(* IEC 61131-3 sources: iolink/src/types/serialization/Simatic.Ax.IOLink/BigEndian, 4 files *)

(* ---- BlockDefinition.st ---- *)
// This is generated code. *** DO NOT MODIFY ***

NAMESPACE Simatic.Ax.iolink
FUNCTION SerializeBig : UDINT
    VAR_INPUT
        offset : UDINT;
    END_VAR
    VAR_IN_OUT
        value : BlockDefinition;
        buffer : ARRAY[*] OF BYTE;
    END_VAR
    SerializeBig := offset;
    SerializeBig := System.Serialization.SerializeBig(offset := SerializeBig, value := value.BlockNoDefinition, buffer := buffer);
    SerializeBig := System.Serialization.SerializeBig(offset := SerializeBig, value := value.Channel, buffer := buffer);
    SerializeBig := System.Serialization.SerializeBig(offset := SerializeBig, value := value.BlockType, buffer := buffer);
    SerializeBig := System.Serialization.SerializeBig(offset := SerializeBig, value := value.Version, buffer := buffer);
    SerializeBig := System.Serialization.SerializeBig(offset := SerializeBig, value := value.ByteLength, buffer := buffer);
END_FUNCTION

FUNCTION DeserializeBig : UDINT
    VAR_INPUT
        offset : UDINT;
        buffer : ARRAY[*] OF BYTE;
    END_VAR
    VAR_IN_OUT
        value : BlockDefinition;
    END_VAR
    DeserializeBig := offset;
    DeserializeBig := System.Serialization.DeserializeBig(offset := DeserializeBig, value := value.BlockNoDefinition, buffer := buffer);
    DeserializeBig := System.Serialization.DeserializeBig(offset := DeserializeBig, value := value.Channel, buffer := buffer);
    DeserializeBig := System.Serialization.DeserializeBig(offset := DeserializeBig, value := value.BlockType, buffer := buffer);
    DeserializeBig := System.Serialization.DeserializeBig(offset := DeserializeBig, value := value.Version, buffer := buffer);
    DeserializeBig := System.Serialization.DeserializeBig(offset := DeserializeBig, value := value.ByteLength, buffer := buffer);
END_FUNCTION
END_NAMESPACE

(* ---- DeviceHeader.st ---- *)
// This is generated code. *** DO NOT MODIFY ***

NAMESPACE Simatic.Ax.iolink
FUNCTION SerializeBig : UDINT
    VAR_INPUT
        offset : UDINT;
    END_VAR
    VAR_IN_OUT
        value : DeviceHeader;
        buffer : ARRAY[*] OF BYTE;
    END_VAR
    SerializeBig := offset;
    SerializeBig := System.Serialization.SerializeBig(offset := SerializeBig, value := value.crc32, buffer := buffer);
    SerializeBig := System.Serialization.SerializeBig(offset := SerializeBig, value := value.SourceDestAddress, buffer := buffer);
    SerializeBig := System.Serialization.SerializeBig(offset := SerializeBig, value := value.TypeIdent, buffer := buffer);
    SerializeBig := System.Serialization.SerializeBig(offset := SerializeBig, value := value.ByteLength, buffer := buffer);
    SerializeBig := System.Serialization.SerializeBig(offset := SerializeBig, value := value.NoOfBlocks, buffer := buffer);
END_FUNCTION

FUNCTION DeserializeBig : UDINT
    VAR_INPUT
        offset : UDINT;
        buffer : ARRAY[*] OF BYTE;
    END_VAR
    VAR_IN_OUT
        value : DeviceHeader;
    END_VAR
    DeserializeBig := offset;
    DeserializeBig := System.Serialization.DeserializeBig(offset := DeserializeBig, value := value.crc32, buffer := buffer);
    DeserializeBig := System.Serialization.DeserializeBig(offset := DeserializeBig, value := value.SourceDestAddress, buffer := buffer);
    DeserializeBig := System.Serialization.DeserializeBig(offset := DeserializeBig, value := value.TypeIdent, buffer := buffer);
    DeserializeBig := System.Serialization.DeserializeBig(offset := DeserializeBig, value := value.ByteLength, buffer := buffer);
    DeserializeBig := System.Serialization.DeserializeBig(offset := DeserializeBig, value := value.NoOfBlocks, buffer := buffer);
END_FUNCTION
END_NAMESPACE

(* ---- LIOLink_typeJob.st ---- *)
// This is generated code. *** DO NOT MODIFY ***

NAMESPACE Simatic.Ax.IOLink
FUNCTION SerializeBig : UDINT
    VAR_INPUT
        offset : UDINT;
    END_VAR
    VAR_IN_OUT
        value : LIOLink_typeJob;
        buffer : ARRAY[*] OF BYTE;
    END_VAR
    VAR_TEMP
        i : DINT;
    END_VAR
    SerializeBig := offset;
    SerializeBig := System.Serialization.SerializeBig(offset := SerializeBig, value := value.ExtendedFunctionNum, buffer := buffer);
    SerializeBig := System.Serialization.SerializeBig(offset := SerializeBig, value := value.Options, buffer := buffer);
    SerializeBig := System.Serialization.SerializeBig(offset := SerializeBig, value := value.SequenceNo, buffer := buffer);
    FOR i := DINT#0 TO DINT#233 DO
        SerializeBig := System.Serialization.SerializeBig(offset := SerializeBig, value := value.payload[i], buffer := buffer);
    END_FOR;
END_FUNCTION

FUNCTION DeserializeBig : UDINT
    VAR_INPUT
        offset : UDINT;
        buffer : ARRAY[*] OF BYTE;
    END_VAR
    VAR_IN_OUT
        value : LIOLink_typeJob;
    END_VAR
    VAR_TEMP
        i : DINT;
    END_VAR
    DeserializeBig := offset;
    DeserializeBig := System.Serialization.DeserializeBig(offset := DeserializeBig, value := value.ExtendedFunctionNum, buffer := buffer);
    DeserializeBig := System.Serialization.DeserializeBig(offset := DeserializeBig, value := value.Options, buffer := buffer);
    DeserializeBig := System.Serialization.DeserializeBig(offset := DeserializeBig, value := value.SequenceNo, buffer := buffer);
    FOR i := DINT#0 TO DINT#233 DO
        DeserializeBig := System.Serialization.DeserializeBig(offset := DeserializeBig, value := value.payload[i], buffer := buffer);
    END_FOR;
END_FUNCTION
END_NAMESPACE

(* ---- LIOLink_typeReadWrite.st ---- *)
// This is generated code. *** DO NOT MODIFY ***

NAMESPACE Simatic.Ax.IOLink
FUNCTION SerializeBig : UDINT
    VAR_INPUT
        offset : UDINT;
    END_VAR
    VAR_IN_OUT
        value : LIOLink_typeReadWrite;
        buffer : ARRAY[*] OF BYTE;
    END_VAR
    VAR_TEMP
        i : DINT;
    END_VAR
    SerializeBig := offset;
    SerializeBig := Simatic.Ax.IOLink.SerializeBig(offset := SerializeBig, value := value.header, buffer := buffer);
    FOR i := DINT#0 TO DINT#231 DO
        SerializeBig := System.Serialization.SerializeBig(offset := SerializeBig, value := value.data[i], buffer := buffer);
    END_FOR;
END_FUNCTION

FUNCTION DeserializeBig : UDINT
    VAR_INPUT
        offset : UDINT;
        buffer : ARRAY[*] OF BYTE;
    END_VAR
    VAR_IN_OUT
        value : LIOLink_typeReadWrite;
    END_VAR
    VAR_TEMP
        i : DINT;
    END_VAR
    DeserializeBig := offset;
    DeserializeBig := Simatic.Ax.IOLink.DeserializeBig(offset := DeserializeBig, value := value.header, buffer := buffer);
    FOR i := DINT#0 TO DINT#231 DO
        DeserializeBig := System.Serialization.DeserializeBig(offset := DeserializeBig, value := value.data[i], buffer := buffer);
    END_FOR;
END_FUNCTION
END_NAMESPACE
